FUNCTION_BLOCK FB_FIFO_ULINT_Array
VAR_IN_OUT
	a_FIFO		: ARRAY [*] OF ULINT;
END_VAR
VAR_OUTPUT
END_VAR
VAR
	nEntryCount		: DINT;
END_VAR

METHOD AddEntry : BOOL
VAR_INPUT
	nEntry		: ULINT;
END_VAR
VAR
	i : DINT;
END_VAR
IF (LOWER_BOUND(a_FIFO, 1) + nEntryCount - 1) > UPPER_BOUND(a_FIFO, 1) THEN
	AddEntry := FALSE;		//FIFO is full
ELSE
	FOR i := UPPER_BOUND(a_FIFO,1) - 1 TO LOWER_BOUND(a_FIFO,1) BY -1 DO
		a_FIFO[i+1] := a_FIFO[i];
	END_FOR
	
	a_FIFO[LOWER_BOUND(a_FIFO,1)] := nEntry;
	
	nEntryCount := nEntryCount + 1;
	AddEntry := TRUE;
END_IF
END_METHOD

PROPERTY EntryCount : DINT
GET
EntryCount := nEntryCount;
END_GET
END_PROPERTY

PROPERTY LastInValue : ULINT
GET
IF nEntryCount = 0 THEN
	LastInValue := 0;
ELSE
	LastInValue := a_FIFO[LOWER_BOUND(a_FIFO,1)];
END_IF
END_GET
END_PROPERTY

PROPERTY NextOutValue : ULINT
GET
IF nEntryCount = 0 THEN
	NextOutValue := 0;
ELSE
	NextOutValue := a_FIFO[LOWER_BOUND(a_FIFO,1) + nEntryCount - 1];
END_IF
END_GET
END_PROPERTY

METHOD RemoveEntry : BOOL
VAR_INPUT
END_VAR
IF nEntryCount = 0 THEN
	RemoveEntry := FALSE;
ELSE
	IF (LOWER_BOUND(a_FIFO,1) + nEntryCount - 1) <= UPPER_BOUND(a_FIFO,1) THEN
		a_FIFO[LOWER_BOUND(a_FIFO,1) + nEntryCount - 1] := 0;
		nEntryCount := nEntryCount - 1; 
		RemoveEntry := TRUE;
	END_IF
END_IF
END_METHOD

END_FUNCTION_BLOCK

(* stored: Version 1.1.0.1, ProductVersion 3.1.4024.9
   POU FB_FIFO_ULINT_Array: Id {4f4ef72e-1eb2-4af8-9b93-244cd89afa08}, SpecialFunc None
   Folder 01_Properties: Id {04c9ba61-7798-4e4b-9e9c-0cf66549ac83}
   Folder 02_Methods: Id {ea47a859-99ea-4659-bcc8-211e82817563}
   Method AddEntry: Id {72b1a6e6-e200-4a64-8774-4cabb80216f9}
   Property EntryCount: Id {0db0dfc1-6d40-4c1e-976f-e47f07d3373a}
   Get Get: Id {4ebdcc23-4f52-4b54-9c01-6dc9d7c4bdcc}
   Property LastInValue: Id {a42b4702-8e0b-4c25-83bd-8dedd4958155}
   Get Get: Id {742fb16d-6ac5-4a5f-9dfd-0f8c4c1f0fbc}
   Property NextOutValue: Id {5ddcee6a-f44f-4319-b718-5438e8996316}
   Get Get: Id {d7eda0fb-1361-47bf-8a55-99148a192f24}
   Method RemoveEntry: Id {264b1497-e44f-4cb6-9f30-9865215b78c5} *)
